{attribute addProperty BoxType "AX8206-0000-0102-0102"}
{attribute addProperty Id "DeviceDevice_F82A60211620Ch_ACh_A_B17182A2176220Ch_BCh_B_7239D878176220WcStateAT %I*WcState_98A4DF7520.250InfoDataAT %I*InfoData_17277C5A208260"}
{attribute addProperty CRC "2269547550"}
{attribute addProperty SizeInBites "578"}
{attribute addProperty SizeInBytes "72.25"}
TYPE AX8206_23A6453C :
STRUCT
	{attribute addProperty Name "Device"}
	Device : Device_F82A6021;
	{attribute addProperty Name "Ch_A"}
	Ch_A : Ch_A_B17182A2;
	{attribute addProperty Name "Ch_B"}
	Ch_B : Ch_B_7239D878;
	{attribute addProperty Name "WcState"}
	WcState : WcState_98A4DF75;
	{attribute addProperty Name "InfoData"}
	InfoData : InfoData_17277C5A;
END_STRUCT
END_TYPE

(* stored: Version 1.2.0.0, ProductVersion 3.1.4024.9
   DUT AX8206_23A6453C: Id {14136e13-a103-4301-83d3-002c78aeeb9b} *)
